INTERFACE I_SequenceTest EXTENDS I_Base, I_Cyclic

{attribute 'monitoring' := 'call'}
PROPERTY Busy : BOOL
GET
END_GET
END_PROPERTY

METHOD Reset
VAR_INPUT
END_VAR
END_METHOD

METHOD Start
VAR_INPUT
END_VAR
END_METHOD

METHOD Stop
VAR_INPUT
END_VAR
END_METHOD

END_INTERFACE

(* stored: Version 1.1.0.1, ProductVersion 3.1.4026.19
   Itf I_SequenceTest: Id {815f0974-c405-48f6-a3a2-102ffcad06f7}
   Property Busy: Id {9118f4bb-bb00-4632-a7b5-7fdc1f3c4e45}
   Get Get: Id {0cc8aedb-ca8a-4d91-b7fa-8062bf7e669e}
   Method Reset: Id {3501d60d-f409-4c95-8a21-7008e1658fa9}
   Method Start: Id {cc128ce8-d56f-40e3-aa0d-9d8de554a659}
   Method Stop: Id {0db30ca2-3dc7-4757-862d-fd83564b862e} *)
